// Mitsubishi GX Works2 project: k08   PLC: Q02/Q02H

PROGRAM MAIN
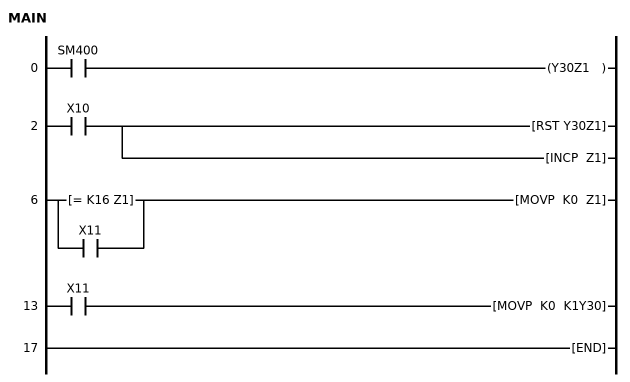
0     LD      SM400
      OUT     Y30Z1
2     LD      X10
      RST     Y30Z1
      INCP    Z1
6     LD=     K16 Z1
      OR      X11
      MOVP    K0 Z1
13    LD      X11
      MOVP    K0 K1Y30
17    END
END_PROGRAM
